Staubli VAL3: insertItem.pgx

public program insertItem(num x_nIndexCopy, num x_nIndexPaste)
begin
  //
  // use to add more elements from the typical one
  //
end
